{attribute 'hide'}
FUNCTION_BLOCK DirectoryEntry_Test EXTENDS TcUnit.FB_TestSuite

IsDirectoryReturnsExpected();

METHOD IsDirectoryReturnsExpected
VAR
	result : BOOL;
	dirEntry : DirectoryEntry('');
END_VAR
TEST('IsDirectoryReturnsExpected');

// @TEST-FIXTURE

// @TEST-RUN
result := dirEntry.IsDirectory;

// @TEST-ASSSERT
AssertTrue(Condition := result, Message := 'IsDirectory did not return TRUE');

TEST_FINISHED();
END_METHOD

END_FUNCTION_BLOCK

(* stored: Version 1.1.0.1, ProductVersion 3.1.4024.9
   POU DirectoryEntry_Test: Id {739998d6-ba93-4aae-a1fe-d62d74083cb7}, SpecialFunc None
   Method IsDirectoryReturnsExpected: Id {64008ed6-09f5-4100-8d0a-feb4d621e890} *)
